// TIA Portal V19 export
TYPE "C301_STU_IF_VEN_TYPIC"
   STRUCT
      CMD_POS { ExternalAccessible := 'False'; ExternalVisible := 'False'; ExternalWritable := 'False'} : Bool;   // Aansturing ventilator positieve richting (Rijrichting)
      CMD_NEG { ExternalAccessible := 'False'; ExternalVisible := 'False'; ExternalWritable := 'False'} : Bool;   // Aansturing ventilator negatieve richting (Tegenrij)
      CMD_RES { ExternalAccessible := 'False'; ExternalVisible := 'False'; ExternalWritable := 'False'} : Bool;   // Reset van de latched storingen
   END_STRUCT;
END_TYPE
